FUNCTION_BLOCK FB_Light IMPLEMENTS __System.IQueryInterface
VAR_INPUT
END_VAR
VAR_OUTPUT
END_VAR
VAR
END_VAR

END_FUNCTION_BLOCK

(* stored: Version 1.1.0.1, ProductVersion 3.1.4024.16
   POU FB_Light: Id {f889c253-9541-476c-bf4c-9f64afbed404}, SpecialFunc None *)
